# EPICS IOC start-up script: test/startup/st.notb-mcs1.iocsh
#Neutron Optics test Bench, E03

epicsEnvSet("MOTOR_PORT",    "$(SM_MOTOR_PORT=MCU1)")

epicsEnvSet("IPADDR",        "$(SM_IPADDR=172.30.32.62)")
epicsEnvSet("IPPORT",        "$(SM_IPPORT=48898)")
epicsEnvSet("AMSNETIDIOC",   "172.30.32.63.1.1")
epicsEnvSet("ASYN_PORT",     "$(SM_ASYN_PORT=MC_CPU1)")
epicsEnvSet("SYSPFX",        "NOTB-MCS1:MC-MCU-01:")
epicsEnvSet("MCUPFX",      "")
epicsEnvSet("PREC",          "$(SM_PREC=3)")
epicsEnvSet("SM_NOAXES",     "4")
epicsEnvSet("ECM_OPTIONS",   "adsPort=852;amsNetIdRemote=5.79.68.164.1.1;amsNetIdLocal=$(AMSNETIDIOC)"

# No poller yet, see ethercatmcStartPoller at the end of the script
epicsEnvSet("ECM_MOVINGPOLLPERIOD", "0")
epicsEnvSet("ECM_IDLEPOLLPERIOD", "0")
< ethercatmcController.iocsh

epicsEnvSet("SYSPFX",        "NOTB-")

#
# Axis 1
#
epicsEnvSet("AXISCONFIG",    "")
epicsEnvSet("AXIS_NAME",    "$(SM_AXIS_NAME=SpGon1:MC-RotX-01:Mtr)")
epicsEnvSet("AXIS_NO",       "$(SM_AXIS_NO=1)")
epicsEnvSet("DESC",          "$(SM_DESC=DESC)")
epicsEnvSet("EGU",           "$(SM_EGU=EGU)")
epicsEnvSet("RAWENCSTEP_ADEL", 0)
epicsEnvSet("RAWENCSTEP_MDEL", 0)
< ethercatmcIndexerAxis.iocsh
< ethercatmcAxisdebug.iocsh

#
# Axis 2
#
epicsEnvSet("AXISCONFIG",    "")
epicsEnvSet("AXIS_NAME",    "$(SM_AXIS_NAME=SpGon1:MC-RotY-01:Mtr)")
epicsEnvSet("AXIS_NO",       "$(SM_AXIS_NO=2)")
epicsEnvSet("DESC",          "$(SM_DESC=DESC)")
epicsEnvSet("EGU",           "$(SM_EGU=EGU)")
epicsEnvSet("RAWENCSTEP_ADEL", 0)
epicsEnvSet("RAWENCSTEP_MDEL", 0)
< ethercatmcIndexerAxis.iocsh
< ethercatmcAxisdebug.iocsh

#
# Axis 3
#
epicsEnvSet("AXISCONFIG",    "")
epicsEnvSet("AXIS_NAME",    "$(SM_AXIS_NAME=SpRot1:MC-RotZ-01:Mtr)")
epicsEnvSet("AXIS_NO",       "$(SM_AXIS_NO=3)")
epicsEnvSet("DESC",          "$(SM_DESC=DESC)")
epicsEnvSet("EGU",           "$(SM_EGU=EGU)")
epicsEnvSet("RAWENCSTEP_ADEL", 0)
epicsEnvSet("RAWENCSTEP_MDEL", 0)
< ethercatmcIndexerAxis.iocsh
< ethercatmcAxisdebug.iocsh

#
# Axis 4
#
epicsEnvSet("AXISCONFIG",    "")
epicsEnvSet("AXIS_NAME",    "$(SM_AXIS_NAME=CamLft:MC-LinZ-01:Mtr)")
epicsEnvSet("AXIS_NO",       "$(SM_AXIS_NO=4)")
epicsEnvSet("DESC",          "$(SM_DESC=DESC)")
epicsEnvSet("EGU",           "$(SM_EGU=EGU)")
epicsEnvSet("RAWENCSTEP_ADEL", 0)
epicsEnvSet("RAWENCSTEP_MDEL", 0)
< ethercatmcIndexerAxis.iocsh
< ethercatmcAxisdebug.iocsh

# Start polling, values are in millisconds
#
epicsEnvSet("MOVINGPOLLPERIOD", "200")
epicsEnvSet("IDLEPOLLPERIOD",   "500")
ethercatmcStartPoller("$(MOTOR_PORT)", "$(MOVINGPOLLPERIOD)", "$(IDLEPOLLPERIOD)")
